(* CoDeSys 2.3 export: WEIGHTBATCHERSUBSTATUS.EXP *)

(* Data type in ENUM *)
TYPE WeightBatcherSubStatus : (WeightBatcherSubStatusNormal:=0, WeightBatcherSubStatusBatching, WeightBatcherSubStatusLoading,
									WeightBatcherSubStatusDischarging, WeightBatcherSubStatusPause, WeightBatcherSubStatusRefStopped,
									WeightBatcherSubStatusRefAlarm, WeightBatcherSubStatusConfErr, WeightBatcherSubStatusForbiddenCommand,
									WeightBatcherSubStatusUnknownCommand, WeightBatcherSubStatusBadCommandParameter);
END_TYPE
